// TIA Portal V19 export
DATA_BLOCK "INTERLOCK DB"   // DB70
{ S7_Optimized_Access := 'FALSE' }
   VAR
      "RO-1 SET PARAMETER" : Struct
         "ORP-301 HH" : Real;
         "ORP-301 H" : Real;
         "pH-301 HIGH" : Real;
         "pH-301 LOW" : Real;
         "pH-302 HIGH" : Real;
         "pH-302 LOW" : Real;
         "CT-301 H" : Real;
         "CT-301 HH" : Real;
         "CT-302 H" : Real;
         "CT-302 HH" : Real;
      END_STRUCT;
      "RO-1 PARAMETER BUFF" : Struct
         "ORP-301 BUFF" : Int;
         "pH-301 BUFF" : Int;
         "pH-302 BUFF" : Int;
         "CT-301 BUFF" : Int;
         "CT-302 BUFF" : Int;
      END_STRUCT;
      "RO-1 SET TIMER" : Struct
         "LPS-301 TIMER SET" : Int;
         "LPS-302 TIMER SET" : Int;
         "HPS-301 TIMER SET" : Int;
         "HPS-302 TIMER SET" : Int;
         "ORP-301 TIMER SET" : Int;
         "CT-301 HIGH TIMER SET" : Int;
         "CT-302 HIGH TIMER SET" : Int;
         "AGLV-301A FLUSH TIME SET" : Int;
         "AGLV-301B FLUSH  TIME SET" : Int;
      END_STRUCT;
      "RO-1 PV TIMER" : Struct
         "LPS-301 TIMER PV" : Int;
         "LPS-302 TIMER PV" : Int;
         "HPS-301 TIMER PV" : Int;
         "HPS-302 TIMER PV" : Int;
         "ORP-301 TIMER PV" : Int;
         "CT-301 HIGH TIMER PV" : Int;
         "CT-302 HIGH TIMER PV" : Int;
         "AGLV-301A FLUSH TIME PV" : Int;
         "AGLV-301B FLUSH  TIME PV" : Int;
      END_STRUCT;
      "RO-2 SET PARAMETER" : Struct
         "pH-401 HIGH" : Real;
         "pH-401 LOW" : Real;
         "pH-402 HIGH" : Real;
         "pH-402 LOW" : Real;
         "CT-401 H" : Real;
         "CT-401 HH" : Real;
         "CT-402 H" : Real;
         "CT-402 HH" : Real;
      END_STRUCT;
      "RO-2 PARAMETER BUFF" : Struct
         "pH-401 BUFF" : Int;
         "pH-402 BUFF" : Int;
         "CT-401 BUFF" : Int;
         "CT-402 BUFF" : Int;
      END_STRUCT;
      "RO-2 SET TIMER" : Struct
         "LPS-401 TIMER SET" : Int;
         "LPS-402 TIMER SET" : Int;
         "HPS-401 TIMER SET" : Int;
         "HPS-402 TIMER SET" : Int;
         "CT-401 HIGH TIMER SET" : Int;
         "CT-402 HIGH TIMER SET" : Int;
         "AGLV-401A FLUSH TIME SET" : Int;
         "AGLV-401B FLUSH  TIME SET" : Int;
      END_STRUCT;
      "RO-2 PV TIMER" : Struct
         "LPS-401 TIMER PV" : Int;
         "LPS-402 TIMER PV" : Int;
         "HPS-401 TIMER PV" : Int;
         "HPS-402 TIMER PV" : Int;
         "CT-401 HIGH TIMER PV" : Int;
         "CT-402 HIGH TIMER PV" : Int;
         "AGLV-401A FLUSH TIME PV" : Int;
         "AGLV-401B FLUSH  TIME PV" : Int;
      END_STRUCT;
      "EDI SET PARAMETER" : Struct
         "PT-501 LOW" : Real;
         "PT-501 HIGH" : Real;
         "PT-502 LOW" : Real;
         "PT-502 HIGH" : Real;
         "PT-503 HIGH" : Real;
         "PT-504 HIGH" : Real;
         "PT-505 HIGH" : Real;
         "PT-506 HIGH" : Real;
         "FIT-501 LOW" : Real;
         "FIT-502 LOW" : Real;
         "FIT-503 LOW" : Real;
         "FIT-504 LOW" : Real;
         "FIT-505 LOW" : Real;
         "FIT-505 HIGH" : Real;
         "FIT-506 LOW" : Real;
         "FIT-506 HIGH" : Real;
         "FIT-507 LOW" : Real;
         "FIT-507 HIGH" : Real;
         "FIT-508 LOW" : Real;
         "FIT-508 HIGH" : Real;
         "pHIT-501 - LOW" : Real;
         "pHIT-501 - High" : Real;
         "pHIT-502 - LOW" : Real;
         "pHIT-502 - High" : Real;
         "RIT-501 HIGH" : Real;
         "RIT-502 HIGH" : Real;
         "RIT-501 LOW" : Real;
         "RIT-502 LOW" : Real;
      END_STRUCT;
      "EDI PARAMETER BUFF" : Struct
         "PT-501 LOW/ HIGH BUFF" : Int;
         "PT-502 LOW / HIGH BUFF" : Int;
         "PT-503 HIGH" : Int;
         "PT-504 HIGH" : Int;
         "PT-505 HIGH" : Int;
         "PT-506 HIGH" : Int;
         "FIT-501 LOW BUFF" : Int;
         "FIT-502 LOW  BUFF" : Int;
         "FIT-503 LOW BUFF" : Int;
         "FIT-504 LOW BUFF" : Int;
         "FIT-505 LOW / HIGH BUFF" : Int;
         "FIT-506 LOW / HIGH BUFF" : Int;
         "FIT-507 LOW / HIGH BUFF" : Int;
         "FIT-508 LOW / HIGH BUFF" : Int;
         "pHIT-501 - LOW / High BUFF" : Int;
         "pHIT-502 - LOW / High BUFF" : Int;
         "RIT-501 HIGH/LOW BUFF" : Int;
         "RIT-502 HIGH/ LOW BUFF" : Int;
      END_STRUCT;
      "EDI SET TIMER" : Struct
         "PT-501 LOW TIMER SET" : Int;
         "PT-501 HIGH TIMER SET" : Int;
         "PT-502 LOW TIMER SET" : Int;
         "PT-502 HIGH TIMER SET" : Int;
         "PT-503 HIGH TIMER SET" : Int;
         "PT-504 HIGH TIMER SET" : Int;
         "PT-505 HIGH TIMER SET" : Int;
         "PT-506 HIGH TIMER SET" : Int;
         "FIT-501 LOW TIMER SET" : Int;
         "FIT-502 LOW TIMER SET" : Int;
         "FIT-503 LOW TIMER SET" : Int;
         "FIT-504 LOW TIMER SET" : Int;
         "FIT-505 LOW TIMER SET" : Int;
         "FIT-505 HIGH TIMER SET" : Int;
         "FIT-506 LOW TIMER SET" : Int;
         "FIT-506 HIGH TIMER SET" : Int;
         "FIT-507 LOW TIMER SET" : Int;
         "FIT-507 HIGH TIMER SET" : Int;
         "FIT-508 LOW TIMER SET" : Int;
         "FIT-508 HIGH TIMER SET" : Int;
         "pHIT-501 - LOW TIMER SET" : Int;
         "pHIT-501 - High TIMER SET" : Int;
         "pHIT-502 - LOW TIMER SET" : Int;
         "pHIT-502 - High TIMER SET" : Int;
         "RIT-501 HIGH TIMER SET" : Int;
         "RIT-502 HIGH TIMER SET" : Int;
      END_STRUCT;
      "EDI PV TIMER" : Struct
         "PT-501 LOW TIMER PV" : Int;
         "PT-501 HIGH TIMER PV" : Int;
         "PT-502 LOW TIMER PV" : Int;
         "PT-502 HIGH TIMER PV" : Int;
         "PT-503 HIGH TIMER PV" : Int;
         "PT-504 HIGH TIMER PV" : Int;
         "PT-505 HIGH TIMER PV" : Int;
         "PT-506 HIGH TIMER PV" : Int;
         "FIT-501 LOW TIMER PV" : Int;
         "FIT-502 LOW TIMER PV" : Int;
         "FIT-503 LOW TIMER PV" : Int;
         "FIT-504 LOW TIMER PV" : Int;
         "FIT-505 LOW TIMER PV" : Int;
         "FIT-505 HIGH TIMER PV" : Int;
         "FIT-506 LOW TIMER PV" : Int;
         "FIT-506 HIGH TIMER PV" : Int;
         "FIT-507 LOW TIMER PV" : Int;
         "FIT-507 HIGH TIMER PV" : Int;
         "FIT-508 LOW TIMER PV" : Int;
         "FIT-508 HIGH TIMER PV" : Int;
         "pHIT-501 - LOW TIMER PV" : Int;
         "pHIT-501 - High TIMER PV" : Int;
         "pHIT-502 - LOW TIMER PV" : Int;
         "pHIT-502 - High TIMER PV" : Int;
         "RIT-501 HIGH TIMER PV" : Int;
         "RIT-502 HIGH TIMER PV" : Int;
      END_STRUCT;
   END_VAR
BEGIN
END_DATA_BLOCK
